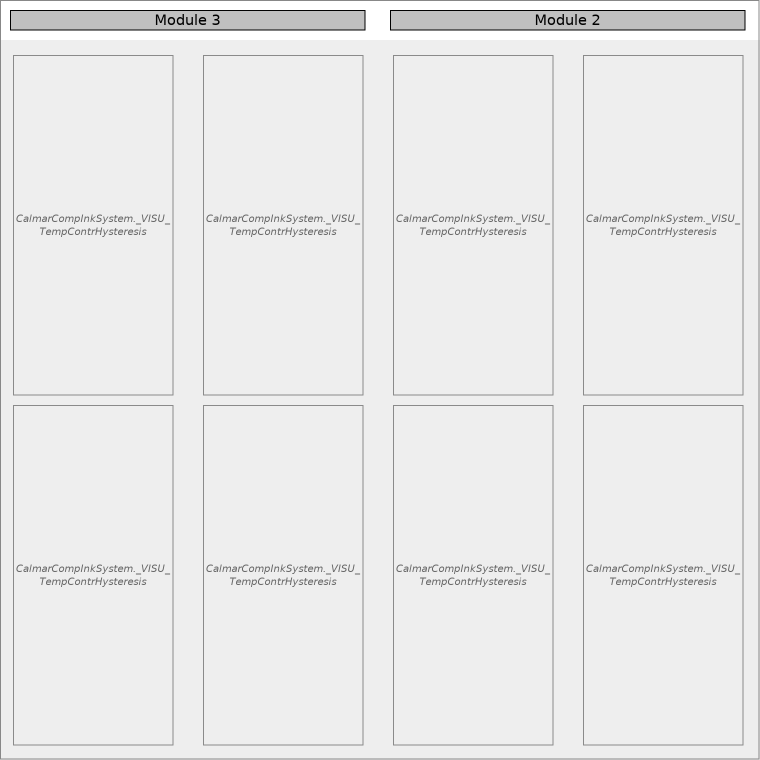
VISUALIZATION VISU_TEMPERATUR  // 760x760
    Rectangle (0,40 760x720)
    Frame (203,55 160x340)
        shows CalmarCompInkSystem._VISU_TempContrHysteresis(m_Inst_Fb := PRG_INK.fb_TempControllerHys[3])
    Frame (393,55 160x340)
        shows CalmarCompInkSystem._VISU_TempContrHysteresis(m_Inst_Fb := PRG_INK.fb_TempControllerHys[2])
    Frame (583,55 160x340)
        shows CalmarCompInkSystem._VISU_TempContrHysteresis(m_Inst_Fb := PRG_INK.fb_TempControllerHys[1])
    Frame (13,55 160x340)
        shows CalmarCompInkSystem._VISU_TempContrHysteresis(m_Inst_Fb := PRG_INK.fb_TempControllerHys[4])
    Frame (203,405 160x340)
        shows CalmarCompInkSystem._VISU_TempContrHysteresis(m_Inst_Fb := PRG_INK.fb_TempControllerHys[7])
    Frame (393,405 160x340)
        shows CalmarCompInkSystem._VISU_TempContrHysteresis(m_Inst_Fb := PRG_INK.fb_TempControllerHys[6])
    Frame (583,405 160x340)
        shows CalmarCompInkSystem._VISU_TempContrHysteresis(m_Inst_Fb := PRG_INK.fb_TempControllerHys[5])
    Frame (13,405 160x340)
        shows CalmarCompInkSystem._VISU_TempContrHysteresis(m_Inst_Fb := PRG_INK.fb_TempControllerHys[8])
    Rectangle (10,10 355x20), "Module 3"
    Rectangle (390,10 355x20), "Module 2"
END_VISUALIZATION

(* stored: Version 1.1.0.1, ProductVersion 3.1.4024.9
   Visu VISU_TEMPERATUR: Id {92f9401b-07ff-476a-83b3-89c27571f116} *)
